// TIA Portal V20 export
VAR_GLOBAL   // PLC tag table "LNK_Const_Gen"
END_VAR
VAR_GLOBAL CONSTANT   // user constants
   LNK_MAGIC : Word := 16#4753;   // FRAME header magic 'GS' / FRAME 헤더 매직 'GS'
   LNK_VERSION : USInt := 1;   // FRAME header version / FRAME 헤더 버전
   LNK_FMT_JSON : USInt := 1;   // Payload format JSON / 페이로드 포맷 JSON
   LNK_FMT_BIN : USInt := 2;   // Payload format BIN (Serialize) / 페이로드 포맷 BIN (Serialize)
   LNK_HDR_LEN : DInt := 16;   // FRAME header length (bytes) / FRAME 헤더 길이 (B)
   LNK_MAX_PAYLOAD : DInt := 8176;   // PLC receive payload / line max (bytes) / PLC 수신 페이로드 / 줄 최대 (B)
   LNK_MSG_HELLO : UInt := 1;   // Message id Hello (LNK_Hello) / 메시지 ID Hello
   LNK_MSG_HEARTBEAT : UInt := 2;   // Message id Heartbeat (no payload) / 메시지 ID Heartbeat (페이로드 없음)
   LNK_MSG_MEASLOG : UInt := 10;   // Message id MeasLog (LGR_MeasureLog) / 메시지 ID MeasLog
   LNK_MSG_STATUS : UInt := 11;   // Message id Status (LNK_GR_Status) / 메시지 ID Status
   LNK_MSG_COMMAND : UInt := 20;   // Message id Command (LGR_Interface_GR_Command) / 메시지 ID Command
   LNK_MSG_COMMANDRESULT : UInt := 21;   // Message id CommandResult (LGR_Command_Response) / 메시지 ID CommandResult
   LNK_MSG_ACK : UInt := 30;   // Message id Ack (LNK_Ack) / 메시지 ID Ack
   LNK_SIG_HELLO : DWord := 16#BFAD9982;   // UDT signature LNK_Hello / UDT 시그니처 LNK_Hello
   LNK_SIG_MEASLOG : DWord := 16#DC0B3DF9;   // UDT signature LGR_MeasureLog / UDT 시그니처 LGR_MeasureLog
   LNK_SIG_STATUS : DWord := 16#2FE5346B;   // UDT signature LNK_GR_Status / UDT 시그니처 LNK_GR_Status
   LNK_SIG_COMMAND : DWord := 16#3B38A0EF;   // UDT signature LGR_Interface_GR_Command / UDT 시그니처 LGR_Interface_GR_Command
   LNK_SIG_COMMANDRESULT : DWord := 16#6D851FD2;   // UDT signature LGR_Command_Response / UDT 시그니처 LGR_Command_Response
   LNK_SIG_ACK : DWord := 16#FF5482FF;   // UDT signature LNK_Ack / UDT 시그니처 LNK_Ack
   LNK_LEN_HELLO : DInt := 28;   // Serialized size LNK_Hello (bytes) / 직렬화 크기 LNK_Hello (B)
   LNK_LEN_MEASLOG : DInt := 236;   // Serialized size LGR_MeasureLog (bytes) / 직렬화 크기 LGR_MeasureLog (B)
   LNK_LEN_STATUS : DInt := 220;   // Serialized size LNK_GR_Status (bytes) / 직렬화 크기 LNK_GR_Status (B)
   LNK_LEN_COMMAND : DInt := 186;   // Serialized size LGR_Interface_GR_Command (bytes) / 직렬화 크기 LGR_Interface_GR_Command (B)
   LNK_LEN_COMMANDRESULT : DInt := 174;   // Serialized size LGR_Command_Response (bytes) / 직렬화 크기 LGR_Command_Response (B)
   LNK_LEN_ACK : DInt := 48;   // Serialized size LNK_Ack (bytes) / 직렬화 크기 LNK_Ack (B)
   LNK_JMAX_HELLO : DInt := 236;   // Max JSON envelope length Hello (bytes) / JSON 엔벨로프 최대 길이 Hello (B)
   LNK_JMAX_MEASLOG : DInt := 1693;   // Max JSON envelope length MeasLog (bytes) / JSON 엔벨로프 최대 길이 MeasLog (B)
   LNK_JMAX_STATUS : DInt := 1905;   // Max JSON envelope length Status (bytes) / JSON 엔벨로프 최대 길이 Status (B)
   LNK_JMAX_COMMAND : DInt := 2448;   // Max JSON envelope length Command (bytes) / JSON 엔벨로프 최대 길이 Command (B)
   LNK_JMAX_COMMANDRESULT : DInt := 2418;   // Max JSON envelope length CommandResult (bytes) / JSON 엔벨로프 최대 길이 CommandResult (B)
   LNK_JMAX_ACK : DInt := 347;   // Max JSON envelope length Ack (bytes) / JSON 엔벨로프 최대 길이 Ack (B)
   LNK_ERR_OK : Int := 0;   // Link error: OK / 링크 오류: 정상
   LNK_ERR_BAD_MAGIC : Int := 1;   // Link error: bad FRAME magic / 링크 오류: FRAME 매직 불일치
   LNK_ERR_BAD_VERSION : Int := 2;   // Link error: bad FRAME version / 링크 오류: FRAME 버전 불일치
   LNK_ERR_UNKNOWN_TYPE : Int := 3;   // Link error: unknown message type / 링크 오류: 알 수 없는 메시지
   LNK_ERR_SIG_MISMATCH : Int := 4;   // Link error: BIN layout signature mismatch / 링크 오류: BIN 시그니처 불일치
   LNK_ERR_BAD_LENGTH : Int := 5;   // Link error: bad length / 링크 오류: 길이 오류
   LNK_ERR_PARSE : Int := 6;   // Link error: parse error / 링크 오류: 파싱 오류
   LNK_ERR_FORMAT_NOT_ALLOWED : Int := 7;   // Link error: format not allowed (BIN over NDJSON) / 링크 오류: 허용되지 않는 포맷 (NDJSON 위 BIN)
   LNK_ERR_DIR_NOT_ALLOWED : Int := 8;   // Link error: direction not allowed / 링크 오류: 허용되지 않는 방향
   LNK_ERR_BUSY : Int := 9;   // Link error: busy / 링크 오류: 처리 중
   LNK_ERR_NO_PENDING : Int := 10;   // Link error: nothing pending / 링크 오류: 대기 항목 없음
   LNK_MSG_TRACECFG : UInt := 40;   // Message id TraceCfg (LNK_TraceCfg)
   LNK_MSG_TRACE : UInt := 41;   // Message id Trace (LNK_Trace)
   LNK_SIG_TRACECFG : DWord := 16#76E981D2;   // UDT signature LNK_TraceCfg
   LNK_SIG_TRACE : DWord := 16#DA67BF12;   // UDT signature LNK_Trace
   LNK_LEN_TRACECFG : DInt := 330;   // Serialized size LNK_TraceCfg (bytes)
   LNK_LEN_TRACE : DInt := 8160;   // Serialized size LNK_Trace (bytes)
   LNK_JMAX_TRACECFG : DInt := 2316;   // Max JSON envelope length TraceCfg (bytes)
   LNK_REGISTRY_HASH : DWord := 16#8E7B313C;   // Message registry hash (crc32, wire-spec 5)
END_VAR
